FUNCTION_BLOCK Wago1405_6 (* Service Interface Function Block Type *)
  (* Standard: 61499-2; Description: Copyright (c) 2018 fortiss GmbH This program and the accompanying materials are made available under the terms of the Eclipse Public License 2.0 which is available at https://www.eclipse.org/legal/epl-2.0/ SPDX-License-Identifier: EPL-2.0 *)
  (* Version 1.0, 2018-12-05, Jose Cabral *)
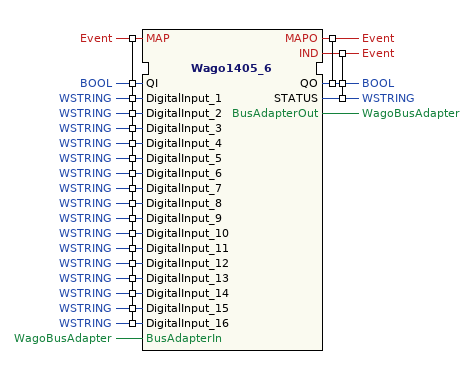
  EVENT_INPUT
    MAP WITH DigitalInput_1, DigitalInput_2, DigitalInput_5, DigitalInput_3, DigitalInput_4, DigitalInput_6, DigitalInput_7, DigitalInput_8, DigitalInput_9, DigitalInput_10, DigitalInput_11, DigitalInput_12, DigitalInput_13, DigitalInput_14, DigitalInput_15, DigitalInput_16, QI; (* Map Pins *)
  END_EVENT
  EVENT_OUTPUT
    MAPO WITH QO; (* Confirm Pin Mapping *)
    IND WITH QO, STATUS; (* Indication from Resource *)
  END_EVENT
  VAR_INPUT
    QI : BOOL; (* Event Input Qualifier *)
    DigitalInput_1 : WSTRING;
    DigitalInput_2 : WSTRING;
    DigitalInput_3 : WSTRING;
    DigitalInput_4 : WSTRING;
    DigitalInput_5 : WSTRING;
    DigitalInput_6 : WSTRING;
    DigitalInput_7 : WSTRING;
    DigitalInput_8 : WSTRING;
    DigitalInput_9 : WSTRING;
    DigitalInput_10 : WSTRING;
    DigitalInput_11 : WSTRING;
    DigitalInput_12 : WSTRING;
    DigitalInput_13 : WSTRING;
    DigitalInput_14 : WSTRING;
    DigitalInput_15 : WSTRING;
    DigitalInput_16 : WSTRING;
  END_VAR
  VAR_OUTPUT
    QO : BOOL; (* Event Output Qualifier *)
    STATUS : WSTRING; (* Service Status *)
  END_VAR
  SOCKETS
    BusAdapterIn : WagoBusAdapter;
  END_SOCKETS
  PLUGS
    BusAdapterOut : WagoBusAdapter;
  END_PLUGS
END_FUNCTION_BLOCK
